	fbGetInputNotification(	bEnable := TRUE,
							eEventScheme := eEventScheme,
							nAddressInfo1 := nAddressInfo01,
							nAddressInfo2 := nAddressInfo02,
							nEventInfo => nInputValue);
	CASE fbGetInputNotification.nEventInfo OF
		0: sInputValue := 'Push button released';
		1: sInputValue := 'Push button pressed';
		2: sInputValue := 'Short press';
		5: sInputValue := 'Double press';
		9: sInputValue := 'Long press start';
		11: sInputValue := 'Long press repeat';
		12: sInputValue := 'Long press stop';
		14: sInputValue := 'Button free';
		15: sInputValue := 'Button stuck';
	END_CASE
{endregion}
{region "Read"}
5:
{region "Start Qiescent Mode"}
	fb103StartQuiescentMode(bStart := TRUE,
							eAddressType := Tc3_DALI.E_DALIAddressType.Broadcast,
							eCommandPriority := Tc3_DALI.E_DALICommandPriority.Middle);
	IF (NOT fb103StartQuiescentMode.bBusy) THEN
		fb103StartQuiescentMode(bStart := FALSE);
		nStep := 10;
	END_IF
{endregion}
10:
{region "Query Instance Error"}
	fb103QueryInstanceError(bStart := TRUE,
							nAddress := nAddress,
							eAddressType := Tc3_DALI.E_DALIAddressType.Short,
							nInstanceAddress := nInstanceAddress,
							eInstanceAddressType := Tc3_DALI.E_DALIInstanceAddressType.InstanceNumber,
							eCommandPriority := Tc3_DALI.E_DALICommandPriority.Middle,
							nInstanceError => nInstanceError);
	IF (NOT fb103QueryInstanceError.bBusy) THEN
		fb103QueryInstanceError(bStart := FALSE);
		nStep := 20;
	END_IF
{endregion}
20:
{region "Query Instance Status"}
	fb103QueryInstanceStatus(	bStart := TRUE,
								nAddress := nAddress,
								eAddressType := Tc3_DALI.E_DALIAddressType.Short,
								nInstanceAddress := nInstanceAddress,
								eInstanceAddressType := Tc3_DALI.E_DALIInstanceAddressType.InstanceNumber,
								eCommandPriority := Tc3_DALI.E_DALICommandPriority.Middle);
	IF (NOT fb103QueryInstanceStatus.bBusy) THEN
		fb103QueryInstanceStatus(bStart := FALSE);
		IF (fb103QueryInstanceStatus.nInstanceStatus.1) THEN
			bEnable := TRUE;
		END_IF
		nStep := 30;
	END_IF
30:
{region "Query Resolution"}
	fb103QueryResolution(	bStart := TRUE,
							nAddress := nAddress,
							eAddressType := Tc3_DALI.E_DALIAddressType.Short,
							nInstanceAddress := nInstanceAddress,
							eInstanceAddressType := Tc3_DALI.E_DALIInstanceAddressType.InstanceNumber,
							eCommandPriority := Tc3_DALI.E_DALICommandPriority.Middle,
							nResolution => nResolution);
	IF (NOT fb103QueryResolution.bBusy) THEN
		fb103QueryResolution(bStart := FALSE);
		nStep := 40;
	END_IF
{endregion}
40:
{region "Query Input Value"}
	fb103QueryInputValue(	bStart := TRUE,
							nAddress := nAddress,
							eAddressType := Tc3_DALI.E_DALIAddressType.Short,
							nInstanceAddress := nInstanceAddress,
							eInstanceAddressType := Tc3_DALI.E_DALIInstanceAddressType.InstanceNumber,
							eCommandPriority := Tc3_DALI.E_DALICommandPriority.Middle,
							nResolution := nResolution);
	IF (NOT fb103QueryInputValue.bBusy) THEN
		fb103QueryInputValue(bStart := FALSE);
		CASE fb103QueryInputValue.nInputValue OF
			0: sInputValue := 'Push button released';
			1: sInputValue := 'Push button pressed';
			2: sInputValue := 'Short press';
			5: sInputValue := 'Double press';
			9: sInputValue := 'Long press start';
			11: sInputValue := 'Long press repeat';
			12: sInputValue := 'Long press stop';
			14: sInputValue := 'Button free';
			15: sInputValue := 'Button stuck';
		END_CASE
		nStep := 50;
	END_IF
{endregion}
50:
{region "Query Event Scheme"}
	fb103QueryEventScheme(	bStart := TRUE,
							nAddress := nAddress,
							eAddressType := Tc3_DALI.E_DALIAddressType.Short,
							nInstanceAddress := nInstanceAddress,
							eInstanceAddressType := Tc3_DALI.E_DALIInstanceAddressType.InstanceNumber,
							eCommandPriority := Tc3_DALI.E_DALICommandPriority.Middle,
							eEventScheme => eEventScheme);
	IF (NOT fb103QueryEventScheme.bBusy) THEN
		fb103QueryEventScheme(bStart := FALSE);
		nStep := 60;
	END_IF
{endregion}
60:
{region "Query Event Filter"}
	fb103QueryEventFilter(	bStart := TRUE,
							nAddress := nAddress,
							eAddressType := Tc3_DALI.E_DALIAddressType.Short,
							nInstanceAddress := nInstanceAddress,
							eInstanceAddressType := Tc3_DALI.E_DALIInstanceAddressType.InstanceNumber,
							eCommandPriority := Tc3_DALI.E_DALICommandPriority.Middle,
							nEventFilter => nEventFilter);
	IF (NOT fb103QueryEventFilter.bBusy) THEN
		fb103QueryEventFilter(bStart := FALSE);
		bButtonReleased := nEventFilter.0;
		bButtonPressed := nEventFilter.1;
		bShortPress := nEventFilter.2;
		bDoublePress := nEventFilter.3;
		bLongPressStart := nEventFilter.4;
		bLongPressRepeat := nEventFilter.5;
		bLongPressStop := nEventFilter.6;
		bButtonStuck := nEventFilter.7;
		nStep := 70;
	END_IF
{endregion}
70:
{region "Query Repeat Timer"}
	fb301QueryRepeatTimer(	bStart := TRUE,
							nAddress := nAddress,
							eAddressType := Tc3_DALI.E_DALIAddressType.Short,
							nInstanceAddress := nInstanceAddress,
							eInstanceAddressType := Tc3_DALI.E_DALIInstanceAddressType.InstanceNumber,
							eCommandPriority := Tc3_DALI.E_DALICommandPriority.Middle);
	nRepeat := (fb301QueryRepeatTimer.nRepeat * 20);
	IF (NOT fb301QueryRepeatTimer.bBusy) THEN
		fb301QueryRepeatTimer(bStart := FALSE);
		nStep := 80;
	END_IF
{endregion}
80:
{region "Query Stuck Timer"}
	fb301QueryStuckTimer(	bStart := TRUE,
							nAddress := nAddress,
							eAddressType := Tc3_DALI.E_DALIAddressType.Short,
							nInstanceAddress := nInstanceAddress,
							eInstanceAddressType := Tc3_DALI.E_DALIInstanceAddressType.InstanceNumber,
							eCommandPriority := Tc3_DALI.E_DALICommandPriority.Middle,
							nStuck => nStuck);
	IF (NOT fb301QueryStuckTimer.bBusy) THEN
		fb301QueryStuckTimer(bStart := FALSE);
		nStep := 90;
	END_IF
{endregion}
90:
{region "Query Short Timer"}
	fb301QueryShortTimer(	bStart := TRUE,
							nAddress := nAddress,
							eAddressType := Tc3_DALI.E_DALIAddressType.Short,
							nInstanceAddress := nInstanceAddress,
							eInstanceAddressType := Tc3_DALI.E_DALIInstanceAddressType.InstanceNumber,
							eCommandPriority := Tc3_DALI.E_DALICommandPriority.Middle);
	nShort := (fb301QueryShortTimer.nShort * 20);
	IF (NOT fb301QueryShortTimer.bBusy) THEN
		fb301QueryShortTimer(bStart := FALSE);
		nStep := 95;
	END_IF
{endregion}
95:
{region "Query Short Timer Min"}
	fb301QueryShortTimerMin(bStart := TRUE,
							nAddress := nAddress,
							eAddressType := Tc3_DALI.E_DALIAddressType.Short,
							nInstanceAddress := nInstanceAddress,
							eInstanceAddressType := Tc3_DALI.E_DALIInstanceAddressType.InstanceNumber,
							eCommandPriority := Tc3_DALI.E_DALICommandPriority.Middle);
	nShortMin := (fb301QueryShortTimerMin.nShortMin * 20);
	IF (NOT fb301QueryShortTimerMin.bBusy) THEN
		fb301QueryShortTimerMin(bStart := FALSE);
		nStep := 100;
	END_IF
{endregion}
100:
{region "Query Double Timer"}
	fb301QueryDoubleTimer(	bStart := TRUE,
							nAddress := nAddress,
							eAddressType := Tc3_DALI.E_DALIAddressType.Short,
							nInstanceAddress := nInstanceAddress,
							eInstanceAddressType := Tc3_DALI.E_DALIInstanceAddressType.InstanceNumber,
							eCommandPriority := Tc3_DALI.E_DALICommandPriority.Middle);
	nDouble := (fb301QueryDoubleTimer.nDouble * 20);
	IF (NOT fb301QueryDoubleTimer.bBusy) THEN
		fb301QueryDoubleTimer(bStart := FALSE);
		nStep := 105;
	END_IF
{endregion}
105:
{region "Query Double Timer"}
	fb301QueryDoubleTimerMin(	bStart := TRUE,
								nAddress := nAddress,
								eAddressType := Tc3_DALI.E_DALIAddressType.Short,
								nInstanceAddress := nInstanceAddress,
								eInstanceAddressType := Tc3_DALI.E_DALIInstanceAddressType.InstanceNumber,
								eCommandPriority := Tc3_DALI.E_DALICommandPriority.Middle);
	nDoubleMin := (fb301QueryDoubleTimerMin.nDoubleMin * 20);
	IF (NOT fb301QueryDoubleTimerMin.bBusy) THEN
		fb301QueryDoubleTimerMin(bStart := FALSE);
		nStep := 110;
	END_IF
{endregion}
110:
{region "Query Event Priority"}
	fb103QueryEventPriority(bStart := TRUE,
							nAddress := nAddress,
							eAddressType := Tc3_DALI.E_DALIAddressType.Short,
							nInstanceAddress := nInstanceAddress,
							eInstanceAddressType := Tc3_DALI.E_DALIInstanceAddressType.InstanceNumber,
							eCommandPriority := Tc3_DALI.E_DALICommandPriority.Middle,
							eEventPriority => eEventPriority);
	IF (NOT fb103QueryEventPriority.bBusy) THEN
		fb103QueryEventPriority(bStart := FALSE);
		nStep := 120;
	END_IF 
{endregion}
120:
{region "Stop Qiescent Mode"}
	fb103StopQuiescentMode(	bStart := TRUE,
							eAddressType := Tc3_DALI.E_DALIAddressType.Broadcast,
							eCommandPriority := Tc3_DALI.E_DALICommandPriority.Middle);
	IF (NOT fb103StopQuiescentMode.bBusy) THEN
		fb103StopQuiescentMode(	bStart := FALSE);
		nStep := 0;
	END_IF
{endregion}
{endregion}
{region "Write"}
1000:
{region "Enable or Disable Instance"}
	IF (bEnable) THEN
		fb103EnableInstance(bStart := TRUE,
							nAddress := nAddress,
							eAddressType := Tc3_DALI.E_DALIAddressType.Short,
							nInstanceAddress := nInstanceAddress,
							eInstanceAddressType := Tc3_DALI.E_DALIInstanceAddressType.InstanceNumber,
							eCommandPriority := Tc3_DALI.E_DALICommandPriority.Middle);
		IF (NOT fb103EnableInstance.bBusy) THEN
			fb103EnableInstance(bStart := FALSE);
			nStep := 1010;
		END_IF
	ELSE
		fb103DisableInstance(	bStart := TRUE,
								nAddress := nAddress,
								eAddressType := Tc3_DALI.E_DALIAddressType.Short,
								nInstanceAddress := nInstanceAddress,
								eInstanceAddressType := Tc3_DALI.E_DALIInstanceAddressType.InstanceNumber,
								eCommandPriority := Tc3_DALI.E_DALICommandPriority.Middle);
		IF (NOT fb103DisableInstance.bBusy) THEN
			fb103DisableInstance(bStart := FALSE);
			nStep := 0;
		END_IF
	END_IF
{endregion}
1010:
{region "Set Event Scheme"}
	fb103SetEventScheme(bStart := TRUE,
						nAddress := nAddress,
						eAddressType := Tc3_DALI.E_DALIAddressType.Short,
						nInstanceAddress := nInstanceAddress,
						eInstanceAddressType := Tc3_DALI.E_DALIInstanceAddressType.InstanceNumber,
						eCommandPriority := Tc3_DALI.E_DALICommandPriority.Middle,
						eEventScheme := eEventScheme);
	IF (NOT fb103SetEventScheme.bBusy) THEN
		fb103SetEventScheme(bStart := FALSE);
		nStep := 1020;
	END_IF
{endregion}
1020:
{region "Set Event Filter"}
	nEventFilter.0 := bButtonReleased;
	nEventFilter.1 := bButtonPressed;
	nEventFilter.2 := bShortPress;
	nEventFilter.3 := bDoublePress;
	nEventFilter.4 := bLongPressStart;
	nEventFilter.5 := bLongPressRepeat;
	nEventFilter.6 := bLongPressStop;
	nEventFilter.7 := bButtonStuck;
	fb103SetEventFilter(bStart := TRUE,
						nAddress := nAddress,
						eAddressType := Tc3_DALI.E_DALIAddressType.Short,
						nInstanceAddress := nInstanceAddress,
						eInstanceAddressType := Tc3_DALI.E_DALIInstanceAddressType.InstanceNumber,
						eCommandPriority := Tc3_DALI.E_DALICommandPriority.Middle,
						nEventFilter := nEventFilter);
	IF (NOT fb103SetEventFilter.bBusy) THEN
		fb103SetEventFilter(bStart := FALSE);
		nStep := 1030;
	END_IF
{endregion}
1030:
{region "Set Repeat Timer"}
	IF (bNoRepeatTimer) THEN
		nStep := 1040;
	ELSE
		fb301SetRepeatTimer(bStart := TRUE,
							nAddress := nAddress,
							eAddressType := Tc3_DALI.E_DALIAddressType.Short,
							nInstanceAddress := nInstanceAddress,
							eInstanceAddressType := Tc3_DALI.E_DALIInstanceAddressType.InstanceNumber,
							eCommandPriority := Tc3_DALI.E_DALICommandPriority.Middle,
							nRepeat := TO_BYTE (nRepeat / 20));
		IF (NOT fb301SetRepeatTimer.bBusy) THEN
			fb301SetRepeatTimer(bStart := FALSE);
			nStep := 1040;
		END_IF
	END_IF
{endregion}
1040:
{region "Set Stuck Timer"}
	IF (bNoStuckTimer) THEN
		nStep := 1050;
	ELSE
		fb301SetStuckTimer(	bStart := TRUE,
							nAddress := nAddress,
							eAddressType := Tc3_DALI.E_DALIAddressType.Short,
							nInstanceAddress := nInstanceAddress,
							eInstanceAddressType := Tc3_DALI.E_DALIInstanceAddressType.InstanceNumber,
							eCommandPriority := Tc3_DALI.E_DALICommandPriority.Middle,
							nStuck := nStuck);
		IF (NOT fb301SetStuckTimer.bBusy) THEN
			fb301SetStuckTimer(bStart := FALSE);
			nStep := 1050;
		END_IF
	END_IF
{endregion}
1050:
{region "Set Short Timer"}
	IF (bNoShortTimer) THEN
		nStep := 1060;
	ELSE
		fb301SetShortTimer(	bStart := TRUE,
							nAddress := nAddress,
							eAddressType := Tc3_DALI.E_DALIAddressType.Short,
							nInstanceAddress := nInstanceAddress,
							eInstanceAddressType := Tc3_DALI.E_DALIInstanceAddressType.InstanceNumber,
							eCommandPriority := Tc3_DALI.E_DALICommandPriority.Middle,
							nShort := TO_BYTE(nShort / 20));
		IF (NOT fb301SetShortTimer.bBusy) THEN
			fb301SetShortTimer(bStart := FALSE);
			nStep := 1060;
		END_IF
	END_IF
{endregion}
1060:
{region "Set Double Timer"}
	IF (bNoDoubleTimer) THEN
		nStep := 1070;
	ELSE
		fb301SetDoubleTimer(bStart := TRUE,
							nAddress := nAddress,
							eAddressType := Tc3_DALI.E_DALIAddressType.Short,
							nInstanceAddress := nInstanceAddress,
							eInstanceAddressType := Tc3_DALI.E_DALIInstanceAddressType.InstanceNumber,
							eCommandPriority := Tc3_DALI.E_DALICommandPriority.Middle,
							nDouble := TO_BYTE(nDouble / 20));
		IF (NOT fb301SetDoubleTimer.bBusy) THEN
			fb301SetDoubleTimer(bStart := FALSE);
			nStep := 1070;
		END_IF
	END_IF
1070:
{region "Set Event Priority"}
	fb103SetEventPriority(	bStart := TRUE,
							nAddress := nAddress,
							eAddressType := Tc3_DALI.E_DALIAddressType.Short,
							nInstanceAddress := nInstanceAddress,
							eInstanceAddressType := Tc3_DALI.E_DALIInstanceAddressType.InstanceNumber,
							eCommandPriority := Tc3_DALI.E_DALICommandPriority.Middle,
							eEventPriority := eEventPriority);
	IF (NOT fb103SetEventPriority.bBusy) THEN
		fb103SetEventPriority(bStart := FALSE);
		nStep := 0;
	END_IF
{endregion}
END_CASE
{endregion}
{endregion}

END_FUNCTION_BLOCK

// ---- POUs/DALI/DALI_Setup/FBs/GearType.TcPOU
FUNCTION GearType : STRING[80]
VAR_INPUT
	nGearType	:	BYTE;
END_VAR
VAR
	i: INT;
	aText	:	ARRAY [0..7] OF STRING[80];
END_VAR

GearType := '';
	aText[0] := 'Output is an electronic switch';
	aText[1] := 'Output is a relay with default open contacts';
	aText[2] := 'Output is a relay with default closed contacts';
	aText[3] := 'Output has a transient suppressor';
	aText[4] := 'Load inrush current limitation is integrated';
	aText[5] := '';
	aText[6] := '';
	aText[7] := '';
FOR i := 0 TO 7 DO
	IF nGearType.0 THEN
		GearType := aText[i];
	ELSE
		GearType := '';
	END_IF
	nGearType := ROR (nGearType,1);
END_FOR

IF (nGearType.1 AND nGearType.2)	THEN 
	GearType := 'Latched Output, the latched state does not change when power is removed';
END_IF

END_FUNCTION

// ---- POUs/DALI/PRGs/EnergyData/P_DALI_Energy_Line.TcPOU
(*
EnergyReporting reads ActiveEnergy (part 252) for all present ballasts on all (configured) DALI-lines where GVL_DALI.g_arrEnergyData[*DALI-line*,*ballast*].bHasEnergyData is TRUE.
Results are stored in GVL_DALI.g_arrEnergyData[*DALI-line*,*ballast*].fActiveEnergy. Energy Data for individual ballasts is NOT persistent.
The engergy sum per DALI-Line (Wh) and Total Energy (kWh) are persistent.

If bCheckActiveEnergy is TRUE, all present ballasts are queried for ActiveEnergy and bHasEnergyData is updated accordingly.
This will result in errors for any ballast that does not comply with part 252.
Errors will not be triggered for activations where bCheckActiveEnergy is FALSE.

After shutdown or download to PLC EnergyReporting is activated automatically internally with bCheckActiveEnergy set to TRUE

EnergyReporting is activated automatically at TOD 0:00, 6:00, 12:00, 18:00 (configurable)

NB:	The priority of commands are set to "middle" internally. Updating all lines will take a couple of minutes to finish, so be patient.
	Other critical commands on the DALI-lines take priotity.
	Add appropriate communication immediately after configuration of a new KL6821 terminal.
	That is, arrfbDALI_EnergyReporting[*DALI-Line*].ipDALICommunication := P_DALI_Background.arrfbKL6821Communication[*DALI-Line*];
*)


PROGRAM P_DALI_Energy_Line
VAR
	arrfbDALI_EnergyReporting	: ARRAY[1..SH_Light.DALI_Param.MAX_DALIV2_LINES] OF FB_DALI_EnergyReporting;
	fbDALI_EnergyDataManagement	: SH_Light.FB_DALI_EnergyDataManagement;
	nNumOfEnergyLines			: BYTE;
	bReadEnergyDataAllLines		: BOOL;
	bReportingDone				: BOOL;
	fbRTrig_ReportingDone		: R_TRIG;
	bRTrigReportingDone			: BOOL;
	
	//Task scheduling
	stLocalSystemTime 		: TIMESTRUCT;
	fbLocalSystemTime 		: FB_LocalSystemTime;
	bGetTime 				: BOOL := TRUE;
	tTimeOut 				: TIME := DEFAULT_ADS_TIMEOUT;
	bLocalSystemTimeValid	: BOOL;
	tzID       				: E_TimeZoneID := eTimeZoneID_Invalid;
	
	tdSystemTime			: TOD;
	btestTodCompare			: BOOL;
	
	
END_VAR
VAR CONSTANT
	tdMidnight						: TOD := TOD#0:0:0;
	tdMorning						: TOD := TOD#6:0:0;
	tdMidDay						: TOD := TOD#12:0:0;
	tdEvening						: TOD := TOD#18:0:0;
	tCheckDuration					: TIME:= T#5S;
	tdTestsum						: TOD := (tdMidnight + tCheckDuration);
END_VAR

VAR PERSISTENT
	arrDaliLineEnergySumWh				: ARRAY[1..SH_Light.DALI_Param.MAX_DALIV2_LINES] OF LREAL;
	fTotalEnergyWh						: LREAL;
	nMaxControlGearOperatingHours		: UINT;
END_VAR


arrfbDALI_EnergyReporting[1].ipDALICommunication := P_DALI_Background.arrfbKL6821Communication[1];
arrfbDALI_EnergyReporting[2].ipDALICommunication := P_DALI_Background.arrfbKL6821Communication[2];
arrfbDALI_EnergyReporting[3].ipDALICommunication := P_DALI_Background.arrfbKL6821Communication[3];
arrfbDALI_EnergyReporting[4].ipDALICommunication := P_DALI_Background.arrfbKL6821Communication[4];
//arrfbDALI_EnergyReporting[5].ipDALICommunication := P_DALI_Background.arrfbKL6821Communication[5];
//arrfbDALI_EnergyReporting[6].ipDALICommunication := P_DALI_Background.arrfbKL6821Communication[6]; // for more update SH_Light.DALI_Param.MAX_DALIV2_LINES

nNumOfEnergyLines := 4;

fbLocalSystemTime(
	sNetID:= '', 
	bEnable:= bGetTime, 
	dwCycle:= 2, // cycle time (in seconds) , Synchronization  every 2 seconds.
	dwOpt:= 1, //Bit 0: If this is set, the Windows system time is additionally synchronized cyclically with the hardware clock (RTC) (corresponds to the function NT_SetTimeToRTCTime).
	tTimeout:= tTimeOut, 
	bValid=> bLocalSystemTimeValid, 
	systemTime=> stLocalSystemTime, 
	tzID=> tzID);
	
tdSystemTime := SYSTEMTIME_TO_TOD(systemTime := stLocalSystemTime);
IF	((tdSystemTime > tdMidnight AND tdSystemTime < (tdMidnight + tCheckDuration)) OR (tdSystemTime > tdMorning AND tdSystemTime < (tdMorning + tCheckDuration)) OR
	(tdSystemTime > tdMidDay AND tdSystemTime < (tdMidDay + tCheckDuration)) OR (tdSystemTime > tdEvening AND tdSystemTime < (tdEvening + tCheckDuration))) THEN
	bReadEnergyDataAllLines := TRUE;
END_IF

fbDALI_EnergyDataManagement(
	NumOfEnergyLines				:= nNumOfEnergyLines,
	bReadEnergyDataAllLines 		:= bReadEnergyDataAllLines,
	arrfbDALI_EnergyReporting		:= arrfbDALI_EnergyReporting,
	arrDaliLineEnergySum			:= arrDaliLineEnergySumWH,
	fTotalEnergyWh					:= fTotalEnergyWh,
	nMaxControlGearOperatingHours	:= nMaxControlGearOperatingHours,
	bReportingDone					=> bReportingDone
);
GVL_AHDataModbus.nTotalEnergy10kWh := TO_UINT(TRUNC(fTotalEnergyWh*EXPT(10,-4)));  //FB_DALI_EnergyDataManagement makes sure only positive values are returned. As so, conversion from REAL to UINT is appropriate
GVL_AHDataModbus.nMaxControlGearOperatingHours := nMaxControlGearOperatingHours;

END_PROGRAM

// ---- POUs/EnOcean/P_EnOcean.TcPOU
PROGRAM P_EnOcean
VAR
	fbKL6581			: FB_KL6581;
	stKL6581_in  AT %I* : KL6581_INPUT;
	stKL6581_out AT %Q*	: KL6581_OUTPUT;
	stKL6581			: STR_KL6581;
	bInitCom			: BOOL := TRUE;
	
	arrEnOcean_Search	: ARRAY [1..8] OF FB_EnOcean_Search;
	nSearchIdx			: BYTE;
	bSerach				: BOOL;
	arrDevices			: ARRAY [1..8] OF INT;
	arrID				: ARRAY [1..8, 0..255] OF DWORD;
	
		//Trykknapper Atrium
	fbAtriumNiveau_Tryk_PladeB				: FB_Rec_RPS_Switch;
	fbAtriumNiveau_Tryk_Sevice				: FB_Rec_RPS_Switch;			

	//Trykknapper på gange

	
	//Trykknapper i rum
	fbRum_4_424_Tryk						: FB_Rec_RPS_Switch;
	fbRum_4_426_Tryk						: FB_Rec_RPS_Switch;
	fbRum_5_441A_Tryk						: FB_Rec_RPS_Switch;
	fbGang_5_441B_Tryk						: FB_Rec_RPS_Switch;
	fbRum_5_444_Tryk						: FB_Rec_RPS_Switch;
	fbRum_5_448A_Tryk						: FB_Rec_RPS_Switch;
	fbRum_5_450_Tryk						: FB_Rec_RPS_Switch;	
	fbRum_5_452_Tryk						: FB_Rec_RPS_Switch;
	fbRum_5_454_Tryk						: FB_Rec_RPS_Switch;
	fbRum_5_411C_Tryk						: FB_Rec_RPS_Switch;
END_VAR

VAR CONSTANT
	byNode_1: BYTE := 1;
	byNode_2: BYTE := 2;
	byNode_3: BYTE := 3;
	byNode_4: BYTE := 4;
	byNode_5: BYTE := 5;
	byNode_6: BYTE := 6;
	byNode_7: BYTE := 7;
	byNode_8: BYTE := 8;
END_VAR


(* Kommunikation mit der KL6581. *)
(* Communication with the KL6581. *)
fbKL6581(
	bInit			:= bInitCom,
	nIdx			:= 2,
	stKL6581_in		:= stKL6581_In,
	stKL6581_out	:= stKL6581_Out,
	bReady			=> ,
	bBusy			=> ,
	bError			=> ,
	iErrorID		=> ,
	str_KL6581		=> stKL6581);

GVL_AHDataModbus.EnOceanError	:= TO_UINT(fbKL6581.iErrorID);
(* Warten bis der Kommunikationsbaustein initialisiert wurde.*)
(* Wait until the communication function block has been initialized. *)
IF (NOT fbKL6581.bReady) THEN
	RETURN;
END_IF

FOR nSearchIdx:= 1 TO 8 DO
	arrEnOcean_Search[nSearchIdx](
		bStart:= TRUE, 
		str_KL6581:= stKL6581 , 
		byNode:= nSearchIdx, 
		bReceive=> , 
		iDevices=>arrDevices[nSearchIdx] , 
		ar_ID=> );
		
		MEMCPY(ADR(arrID[nSearchIdx,0]), ADR(arrEnOcean_Search[nSearchIdx].ar_ID), SIZEOF(arrEnOcean_Search[nSearchIdx].ar_ID)); 
END_FOR

//Gange



//RUM
 //
P_Rum_4_424();
P_Rum_4_426();
P_Rum_5_441A();
P_Gang_5_441B();
P_Rum_5_444();
P_Rum_5_448A();
P_Rum_5_450();
P_Rum_5_452();
P_Rum_5_454();
P_Rum_5_411C();
//AtriumNiveau
A_AtriumNiveau();

ACTION A_AtriumNiveau:
fbAtriumNiveau_Tryk_PladeB(
	str_KL6581:=stKL6581 , 
	byNode:=0, 
	dw_ID:= 16#0029B92D, 
	str_EnOceanSwitch=> GVL_EnOcean.strEnOceanSwitch_AtriumNiveau_PladeB,
	by_Node=> , 
	bReceive=> );

//knap 2 
(*
fbAtriumNiveau_Tryk_Sevice(
	str_KL6581:=stKL6581 , 
	byNode:=0, 
	dw_ID:= 16#00FEE4FE87, 
	str_EnOceanSwitch=> GVL_EnOcean.strEnOceanSwitch_AtriumNiveau_Service, 
	by_Node=> , 
	bReceive=> );
*)
END_ACTION

ACTION P_Gang_5_441B:
fbGang_5_441B_Tryk(
	str_KL6581:=stKL6581 , 
	byNode:=4 , 
	dw_ID:=  16#002A0890, 
	str_EnOceanSwitch=> GVL_EnOcean.strEnOceanSwitch_Gang_5_441B, 
	by_Node=> , 
	bReceive=> );
END_ACTION

ACTION P_Rum_4_424:
fbRum_4_424_Tryk(
	str_KL6581:=stKL6581 , 
	byNode:=2 , 
	dw_ID:= 16#0029AB88, 
	str_EnOceanSwitch=> GVL_EnOcean.strEnOceanSwitch_Rum_4_424, 
	by_Node=> , 
	bReceive=> );
END_ACTION

ACTION P_Rum_4_426:
fbRum_4_426_Tryk(
	str_KL6581:=stKL6581 , 
	byNode:=2 , 
	dw_ID:= 16#0029AAD6, 
	str_EnOceanSwitch=> GVL_EnOcean.strEnOceanSwitch_Rum_4_426, 
	by_Node=> , 
	bReceive=> );
END_ACTION

ACTION P_Rum_5_411C:
fbRum_5_411C_Tryk(
	str_KL6581:=stKL6581 , 
	byNode:=4 , 
	dw_ID:=  16#0029AD43, 
	str_EnOceanSwitch=> GVL_EnOcean.strEnOceanSwitch_Rum_5_411C, 
	by_Node=> , 
	bReceive=> );
END_ACTION

ACTION P_Rum_5_441A:
fbRum_5_441A_Tryk(
	str_KL6581:=stKL6581 , 
	byNode:=4 , 
	dw_ID:=  16#00290EC2, 
	str_EnOceanSwitch=> GVL_EnOcean.strEnOceanSwitch_Rum_5_441A, 
	by_Node=> , 
	bReceive=> );
END_ACTION

ACTION P_Rum_5_444:
fbRum_5_444_Tryk(
	str_KL6581:=stKL6581 , 
	byNode:=4 , 
	dw_ID:=  16#0029B74E, 
	str_EnOceanSwitch=> GVL_EnOcean.strEnOceanSwitch_Rum_5_444, 
	by_Node=> , 
	bReceive=> );
END_ACTION

ACTION P_Rum_5_448A:
fbRum_5_448A_Tryk(
	str_KL6581:=stKL6581 , 
	byNode:=4 , 
	dw_ID:=  16#0029AB8B, 
	str_EnOceanSwitch=> GVL_EnOcean.strEnOceanSwitch_Rum_5_448A, 
	by_Node=> , 
	bReceive=> );
END_ACTION

ACTION P_Rum_5_450:
fbRum_5_450_Tryk(
	str_KL6581:=stKL6581 , 
	byNode:=4 , 
	dw_ID:=  16#0029ABB9, 
	str_EnOceanSwitch=> GVL_EnOcean.strEnOceanSwitch_Rum_5_450, 
	by_Node=> , 
	bReceive=> );
END_ACTION

ACTION P_Rum_5_452:
fbRum_5_452_Tryk(
	str_KL6581:=stKL6581 , 
	byNode:=4 , 
	dw_ID:=  16#0029B8D2, 
	str_EnOceanSwitch=> GVL_EnOcean.strEnOceanSwitch_Rum_5_452, 
	by_Node=> , 
	bReceive=> );
END_ACTION

ACTION P_Rum_5_454:
fbRum_5_454_Tryk(
	str_KL6581:=stKL6581 , 
	byNode:=4 , 
	dw_ID:=  16#0029B75D, 
	str_EnOceanSwitch=> GVL_EnOcean.strEnOceanSwitch_Rum_5_454, 
	by_Node=> , 
	bReceive=> );
END_ACTION

END_PROGRAM

// ---- POUs/MAIN.TcPOU
PROGRAM MAIN
VAR
	nAlive: INT;
	breset: BOOL;
	nDemoVariable : INT;
	nCX8200_State	AT %I*	: UINT;
	P_Rum_6_217: INT;
END_VAR

VAR PERSISTENT
	nDemoVar_Persist: INT;
END_VAR

nAlive:= nAlive + 1;
GVL_AHDataModbus.nCX8200_State_MB := nCX8200_State;

P_SystemDK.M_nCyclic(bReset := breset );
P_DALI_DIAG();
DALI_Commissioning();
P_DALI_Energy_Line();
P_AHModbusComm();


//Gange
P_Gang_4_413();
P_Gang_5_441B();
P_gang_7_401();
P_Gang_4_434A();
P_gang_5_441();


//Rum
P_Rum_4_426();
P_Rum_4_424();

P_rum_5_441A();
P_Rum_5_411C();
P_Rum_5_444();
P_Rum_5_448A();
P_Rum_5_448B();
P_Rum_5_450B();
P_Rum_5_450();
P_Rum_5_452();
P_Rum_5_454();
P_Rum_5_456();


//Testprogrammer
//P_DALI_Energy_Firmware_Test();

END_PROGRAM

// ---- GlobalTextList.TcGTLO
TEXTLIST GlobalTextList
  3955 = ' %5.2f h'
  1376 = ' %d %%'
  307 = ' %d days'
  1111 = '%2.1f  mA'
  102 = '%5.1f W'
  269 = '%5.2f h'
  621 = '%d'
  1617 = '%d %%'
  2081 = '%d days'
  3200 = '%d h'
  1372 = '%d Hz'
  2105 = '%d min'
  2025 = '%d ms'
  1540 = '%d s'
  1613 = '%d V'
  2272 = '%d weeks'
  1359 = '%d °C'
  376 = '%s'
  640 = '0'
  641 = '1'
  661 = '10'
  662 = '11'
  663 = '12'
  999 = '13'
  1000 = '14'
  1001 = '15'
  1002 = '16'
  1003 = '17'
  1004 = '18'
  1005 = '19'
  195 = '2'
  1006 = '20'
  1007 = '21'
  1008 = '22'
  1009 = '23'
  1010 = '24'
  1011 = '25'
  1012 = '26'
  1013 = '27'
  1014 = '28'
  1015 = '29'
  654 = '3'
  1016 = '30'
  1017 = '31'
  1018 = '32'
  1019 = '33'
  1020 = '34'
  1021 = '35'
  1022 = '36'
  1023 = '37'
  1024 = '38'
  1025 = '39'
  655 = '4'
  1026 = '40'
  1027 = '41'
  1028 = '42'
  1029 = '43'
  1030 = '44'
  1031 = '45'
  1032 = '46'
  1033 = '47'
  1034 = '48'
  1035 = '49'
  656 = '5'
  358 = '50'
  359 = '51'
  360 = '52'
  361 = '53'
  362 = '54'
  363 = '55'
  364 = '56'
  365 = '57'
  366 = '58'
  367 = '59'
  657 = '6'
  368 = '60'
  369 = '61'
  370 = '62'
  371 = '63'
  658 = '7'
  659 = '8'
  660 = '9'
  1089 = 'AC-supply possible'
  644 = 'Actual Level:'
  650 = 'Address Type'
  236 = 'Addressing Per Physical Selection Supported'
  1533 = 'Adjustable Emergency Level'
  1175 = 'AM Operation active:'
  1044 = 'AM operation possible'
  1045 = 'Auto Test Capability'
  1799 = 'Battery Charge'
  710 = 'Battery Duration Failure'
  3347 = 'Battery Failure'
  3316 = 'Battery Fully Charged'
  2471 = 'Bit 0'
  379 = 'Bit 1'
  2734 = 'Bit 2'
  2320 = 'Bit 3'
  929 = 'Bit 4'
  2576 = 'Bit 5'
  2065 = 'Bit 6'
  1623 = 'Bit 7'
  6 = 'Bottom Button'
  471 = 'Broadcast'
  482 = 'Button 1'
  720 = 'Button 2'
  515 = 'Button pressed'
  498 = 'Button released'
  527 = 'Button stuck / free'
  3304 = 'Cancel Hold Timer'
  2101 = 'Catch Movement'
  2319 = 'Catching:'
  897 = 'Change Addresses'
  1971 = 'Checkbox'
  372 = 'Choose group:'
  98 = 'Choose scene:'
  1571 = 'Circuit Failure'
  1538 = 'Commands'
  618 = 'Complete new installation \n(all addresses will be removed)'
  807 = 'Control'
  645 = 'Control Gear Failure:'
  445 = 'Current protection active:'
  1716 = 'Current protection device'
  668 = 'Current protection enabled:'
  5 = 'Current Protector Enabled '
  1902 = 'DALI Line:'
  1135 = 'DC-supply possible'
  560 = 'Deadtime Timer:'
  1180 = 'DI1 falling edge'
  1218 = 'DI1 rising edge'
  1726 = 'DI2 falling edge'
  1876 = 'DI2 rising edge'
  519 = 'Dim Dwn'
  63 = 'Dim Up'
  2002 = 'Dimmer Temperature'
  936 = 'Dimming Curve:'
  1317 = 'Dimming method bit 0'
  776 = 'Dimming method bit 1'
  2135 = 'Do not lock process image in case of \nDALI commands from DI1 or DI2'
  4011 = 'Double press'
  1112 = 'Double Timer Min:'
  3936 = 'Double Timer:'
  811 = 'Down'
  594 = 'Down Switch-Off Threshold'
  2357 = 'Down Switch-On Threshold'
  1482 = 'Duration Test Delay Time'
  3527 = 'Duration Test Done And Result Valid'
  3086 = 'Duration Test Failed'
  3077 = 'Duration Test Interval'
  2631 = 'Duration Test Is In Progress'
  2791 = 'Duration Test Max. Delay Exceed'
  1708 = 'Duration Test Request Pending'
  2905 = 'Duration Test Result'
  1759 = 'Emergency Lamp Failure'
  779 = 'Emergency Level'
  3733 = 'Emergency MaxLevel'
  3168 = 'Emergency Min Level'
  1204 = 'Emergency Mode'
  971 = 'Emergency Mode Active'
  1901 = 'Emergency Status'
  486 = 'Enable'
  828 = 'Enable:'
  1982 = 'EventPriority'
  32 = 'EventPriority:'
  494 = 'EventScheme'
  1113 = 'EventScheme:'
  125 = 'Extended Emergency Mode Active'
  1841 = 'Extended Fade Time only valid if Fade Time equals 0!'
  3956 = 'Extended Version'
  649 = 'Fade Running:'
  1074 = 'FadeRate'
  1079 = 'FadeTime'
  1610 = 'Failure Status'
  319 = 'Fast Fade Time:'
  2099 = 'Features'
  672 = 'Features (Read only)'
  206 = 'Features Byte 1'
  377 = 'Features Byte 2'
  2876 = 'Features Byte 3'
  3334 = 'Function Test Delay Time'
  3242 = 'Function Test Done And Result Valid'
  2712 = 'Function Test Failed'
  1801 = 'Function Test Interval'
  1945 = 'Function Test Is In Progress'
  3448 = 'Function Test Max. Delay Exceed'
  165 = 'Function Test Request Pending'
  967 = 'Gang 1.312A'
  256 = 'Gang 1.315'
  906 = 'Gang 1.316'
  207 = 'Gang 2.344'
  66 = 'Gang 2.344A'
  583 = 'Gang 2.350'
  985 = 'Gang 3.362A'
  67 = 'Gang 3.363A'
  173 = 'Gang 3.363B'
  406 = 'Gang 4.308'
  459 = 'Gang 4.330'
  327 = 'Gang 5.338'
  524 = 'Gang 6.310'
  316 = 'Gang 7.301'
  3204 = 'Gear Type'
  1409 = 'GearType'
  815 = 'Go to Scene'
  99 = 'Go to scene'
  468 = 'Group Address'
  2361 = 'Hardwired Inhibit Is Active'
  3553 = 'Hardwired Inhibit Supported'
  2225 = 'Hardwired Switch Is On'
  568 = 'Hold Timer:'
  199 = 'Hysteresis Min:'
  200 = 'Hysteresis:'
  790 = 'Identification Active'
  315 = 'Illuminance Level'
  37 = 'Inhibit'
  3340 = 'Inhibit Mode'
  540 = 'Input Value:'
  544 = 'Instance Error:'
  2895 = 'Instance Number:'
  3047 = 'Integral Control Gear'
  492 = 'Internal DALI power supply disabled'
  1771 = 'K-Bus Watchdog'
  3636 = 'Lamp Emergency Time'
  647 = 'Lamp Failure:'
  2812 = 'Lamp Total Operation Time'
  1521 = 'Leading Edge Mode Running'
  506 = 'LED module integrated'
  2077 = 'Linear Dimming Curve Active'
  2179 = 'Load current can be queried '
  1266 = 'Load Current Overload'
  1355 = 'Load current overload with output \nlevel reduction can be queried'
  306 = 'Load Decrease:'
  1137 = 'Load Increase:'
  2313 = 'Load over-current can be queried'
  2518 = 'Load Over-Current Shutdown'
  1226 = 'Load Rating'
  2963 = 'Load rating can be queried'
  2785 = 'Load unsuitable can be queried'
  1454 = 'Load voltage can be queried'
  516 = 'Load Voltage Out Of Limits'
  1811 = 'Lockable bytes: changeable if "Offset 2" has the Value 85 (0x55).\nFor changing use decimal value.'
  523 = 'Long press repeat'
  507 = 'Long press start'
  511 = 'Long press stop'
  43 = 'Lys Auto'
  444 = 'Lys Rum'
  489 = 'Lys Zone 1'
  2032 = 'Maintained Control Gear'
  2046 = 'Memory Bank:'
  3290 = 'Movement'
  531 = 'na'
  23 = 'Name'
  926 = 'Name of byte in memory bank'
  729 = 'NewAddress'
  588 = 'No Movement'
  1061 = 'Non-logarithmic dimming curve can \nbe selected'
  1795 = 'Normal Mode Active'
  572 = 'Occupied'
  808 = 'Off'
  22 = 'Offset'
  1329 = 'Offset in memory bank'
  726 = 'OldAddress'
  816 = 'On and Step Up'
  1207 = 'Open circuit detection can be queried'
  277 = 'Open Circuit:'
  1375 = 'Open Ciruit (No Load) Detect'
  619 = 'Optical feedback'
  963 = 'Output is current controlled'
  844 = 'Output regulated by current:'
  1545 = 'Parameters'
  2547 = 'Parameters Absolute Input Device'
  1580 = 'Parameters Generic Instance'
  78 = 'Parameters LED'
  309 = 'Parameters Light Sensor'
  556 = 'Parameters Occupancy Sensor'
  465 = 'Parameters Pushbutton Sensor'
  3234 = 'Physical Selection Supported'
  1847 = 'Physical selection supported'
  708 = 'PIR'
  457 = 'PIR status'
  1071 = 'Please check if Current Protector is present \nby reading parameters first.'
  308 = 'Please select the desired Short Address in the table above.'
  1458 = 'Please select the function you need from dropdown above'
  751 = 'Position Event'
  245 = 'Possible Operating Modes'
  719 = 'Power pulse operation'
  1744 = 'Power supply integrated'
  1561 = 'PP Operation active:'
  2321 = 'Prolong Time (30sec / Step)'
  970 = 'PWM Operation active:'
  1882 = 'PWM operation possible'
  1487 = 'Query idle time detection \nenabled'
  701 = 'Query load decrease enabled'
  1351 = 'Query load increase enabled'
  837 = 'Query reduction luminous flux \nregarding thermal overload'
  463 = 'Query short circuit enabled'
  1293 = 'Query thermal switch enabled'
  617 = 'Random Addressing'
  2174 = 'Rated Duration'
  881 = 'Re-Light / Reset Inhibit'
  373 = 'Read'
  1611 = 'Read Only'
  1531 = 'Reads all Fading Parameters'
  768 = 'Real Load Power'
  854 = 'Real load power can be queried'
  810 = 'Recall Max Level'
  809 = 'Recall Min Level'
  186 = 'Ref. Measurement failed:'
  439 = 'Reference System Power'
  2713 = 'Relight Rest Mode Supported'
  580 = 'Repeat'
  470 = 'Repeat Timer:'
  1913 = 'Report Timer:'
  716 = 'Reset Duration Test Done Flag'
  592 = 'Reset Function Test Done Flag'
  2418 = 'Reset inactive process image'
  3150 = 'Reset Lamp Time'
  648 = 'Reset State:'
  2888 = 'Resolution:'
  299 = 'Rest'
  591 = 'Rest Mode Active'
  2001 = 'RMS Load Current'
  784 = 'RMS Load Voltage'
  586 = 'RMS Supply Voltage'
  874 = 'Rum 1.106'
  65 = 'Rum 1.108'
  175 = 'Rum 1.111A'
  924 = 'Rum 1.111C'
  219 = 'Rum 1.111D'
  690 = 'Rum 1.111E'
  912 = 'Rum 1.115'
  126 = 'Rum 1.118'
  215 = 'Rum 1.312A'
  725 = 'Rum 1.318'
  839 = 'Rum 1.319'
  456 = 'Rum 1.320'
  800 = 'Rum 1.321'
  622 = 'Rum 1.322'
  646 = 'Rum 1.323'
  966 = 'Rum 1.324'
  95 = 'Rum 1.325'
  335 = 'Rum 1.326'
  150 = 'Rum 1.327'
  651 = 'Rum 1.328'
  980 = 'Rum 1.330'
  262 = 'Rum 1115'
  642 = 'Rum 2.341'
  978 = 'Rum 2.345'
  736 = 'Rum 2.349'
  593 = 'Rum 2.351'
  122 = 'Rum 2.352'
  27 = 'Rum 2.353'
  41 = 'Rum 2.354'
  697 = 'Rum 2.355'
  826 = 'Rum 2.356'
  561 = 'Rum 2.357'
  415 = 'Rum 3.365'
  981 = 'Rum 3.366'
  865 = 'Rum 3.367'
  212 = 'Rum 3.368'
  921 = 'Rum 3.369'
  329 = 'Rum 3.370'
  2134 = 'Rum 5.356'
  15 = 'Rum 5_352'
  430 = 'Rum 6.310 Sofagruppe'
  348 = 'Rum 6.327'
  891 = 'Rum 6.328'
  11 = 'Rum 6.329'
  72 = 'Rum 6.330B'
  197 = 'Rum 6.331'
  564 = 'Rum 6.333'
  997 = 'Rum 6.337'
  31 = 'Rum 6_330A'
  616 = 'Scan devices by address'
  1036 = 'Scene Level'
  814 = 'Scene:'
  1366 = 'Set Extended Fade Time'
  252 = 'Set Fade Rate'
  1875 = 'Set Fade Time'
  464 = 'Short Address'
  1090 = 'Short Address Range'
  1041 = 'Short Address:'
  34 = 'Short Circuit:'
  503 = 'Short press'
  1516 = 'Short Timer Min:'
  478 = 'Short Timer:'
  2548 = 'Shutdown Invalid Dimming Method'
  1085 = 'Single Short Address'
  395 = 'SP_Lux: %.0f'
  525 = 'SP_Lux: %f'
  615 = 'Start'
  582 = 'Start Duration Test'
  2374 = 'Start Function Test'
  155 = 'Start Identification'
  620 = 'Start with address:'
  2346 = 'State Incandescent Lamp'
  643 = 'Status'
  958 = 'Status Absolute Input Device'
  2506 = 'Status Generic Instance'
  77 = 'Status LED'
  317 = 'Status Light Sensor'
  597 = 'Status Occupancy Sensor'
  536 = 'Status Pushbutton Sensor'
  558 = 'Step Down'
  813 = 'Step Down and Off'
  818 = 'Step Up'
  1193 = 'Stop Test'
  164 = 'Stuck Timer:'
  1256 = 'Supply Frequency'
  2271 = 'Supply frequency can be queried'
  1975 = 'Supply Frequency Out of Limits'
  2505 = 'Supply voltage can be queried'
  2707 = 'Supply Voltage Out Of Limits'
  1042 = 'Switch Off'
  375 = 'Switch On'
  3781 = 'Switched Maintained Control Gear'
  2168 = 'Temperature can be queried'
  2458 = 'Terminal Event'
  1848 = 'Test Execution Timeout'
  849 = 'Test Type A'
  2013 = 'Thermal Overload'
  2042 = 'Thermal Overload with output\nlevel reduction can be queried'
  1108 = 'Thermal Overload:'
  355 = 'Thermal Shut Down:'
  2507 = 'Thermal Shutdown'
  2226 = 'Thermal Shutdown can be queried'
  2733 = 'Threshold Editable'
  305 = 'To'
  973 = 'Top Button'
  136 = 'Trailing Edge ModeRunning'
  475 = 'Unaddressed'
  817 = 'Up'
  3123 = 'Up Switch-Off Threshold'
  1449 = 'Up Switch-On Threshold'
  2521 = 'V%s'
  576 = 'Vacant'
  1205 = 'Value'
  24 = 'Value Dec'
  1435 = 'Value decimal'
  25 = 'Value Hex'
  2231 = 'Value hexadecimal,\nto change use\nvalue decimal'
  374 = 'Write'
  2104 = 'Write\nDimming Curve'
  1047 = 'Write default values'
  490 = 'Write parameters'
END_TEXTLIST

// ---- POUs/Alle_Rum/Gange/Gang_4_434A/Visualization_4_330_1_1_1_1_2.TcVIS
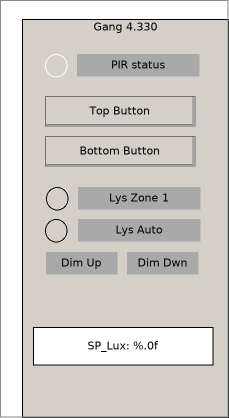
VISUALIZATION Visualization_4_330_1_1_1_1_2  // 229x418
    RoundedRectangle (22,19 207x399), "Gang 4.330"
    Rectangle (33,327 180x38), "SP_Lux: %.0f", text variable: P_Gang_5_135A.arrfbLysGruppe[1].fbLightCtrl.fLuxZone1
    Button (45,96 150x30), "Top Button"
        tap P_Gang_5_135A.bTopButtonZone1_Visu
    Button (45,136 150x30), "Bottom Button"
        tap P_Gang_5_135A.bBottomButtonZone1_Visu
    Ellipse (46,187 22x23), colour toggle: P_Gang_5_135A.fbLys.fbLightCtrl.bOnZone1
    Rectangle (78,187 122x22), "Lys Zone 1"
    Rectangle (46,252 71x22), "Dim Up", colour toggle: P_Gang_5_135A.arrfbLysGruppe[1].fbLightCtrl.bDimUp
    Rectangle (127,252 71x22), "Dim Dwn", colour toggle: P_Gang_5_135A.arrfbLysGruppe[1].fbLightCtrl.bDimDwn
    Ellipse (45,219 22x23), colour toggle: P_Gang_5_135A.arrfbLysGruppe[1].fbLightCtrl.bAutoZone1
    Rectangle (78,219 122x22), "Lys Auto"
    Ellipse (45,54 22x23), colour toggle: P_Gang_5_135A.arrfbLysGruppe[1].fbLightCtrl.bPIR
    Rectangle (77,54 122x22), "PIR status"
END_VISUALIZATION

// ---- POUs/Alle_Rum/Rum_Med_DALI_Pir/Rum_5_450/Visualization_4_330_1_1_1_1_2_1_1_1_3_1.TcVIS
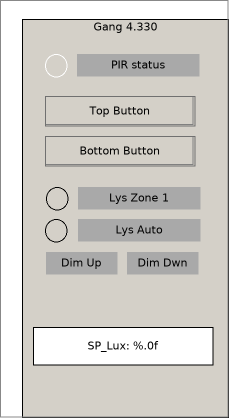
VISUALIZATION Visualization_4_330_1_1_1_1_2_1_1_1_3_1  // 229x418
    RoundedRectangle (22,19 207x399), "Gang 4.330"
    Rectangle (33,327 180x38), "SP_Lux: %.0f", text variable: P_Gang_5_135A.arrfbLysGruppe[1].fbLightCtrl.fLuxZone1
    Button (45,96 150x30), "Top Button"
        tap P_Gang_5_135A.bTopButtonZone1_Visu
    Button (45,136 150x30), "Bottom Button"
        tap P_Gang_5_135A.bBottomButtonZone1_Visu
    Ellipse (46,187 22x23), colour toggle: P_Gang_5_135A.fbLys.fbLightCtrl.bOnZone1
    Rectangle (78,187 122x22), "Lys Zone 1"
    Rectangle (46,252 71x22), "Dim Up", colour toggle: P_Gang_5_135A.arrfbLysGruppe[1].fbLightCtrl.bDimUp
    Rectangle (127,252 71x22), "Dim Dwn", colour toggle: P_Gang_5_135A.arrfbLysGruppe[1].fbLightCtrl.bDimDwn
    Ellipse (45,219 22x23), colour toggle: P_Gang_5_135A.arrfbLysGruppe[1].fbLightCtrl.bAutoZone1
    Rectangle (78,219 122x22), "Lys Auto"
    Ellipse (45,54 22x23), colour toggle: P_Gang_5_135A.arrfbLysGruppe[1].fbLightCtrl.bPIR
    Rectangle (77,54 122x22), "PIR status"
END_VISUALIZATION

// ---- POUs/Alle_Rum/Rum_Med_DALI_Pir/Rum_5_448B/Visualization_4_330_1_1_1_1_2_1.TcVIS
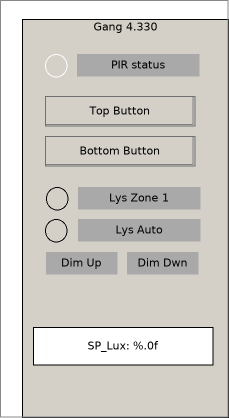
VISUALIZATION Visualization_4_330_1_1_1_1_2_1  // 229x418
    RoundedRectangle (22,19 207x399), "Gang 4.330"
    Rectangle (33,327 180x38), "SP_Lux: %.0f", text variable: P_Gang_5_135A.arrfbLysGruppe[1].fbLightCtrl.fLuxZone1
    Button (45,96 150x30), "Top Button"
        tap P_Gang_5_135A.bTopButtonZone1_Visu
    Button (45,136 150x30), "Bottom Button"
        tap P_Gang_5_135A.bBottomButtonZone1_Visu
    Ellipse (46,187 22x23), colour toggle: P_Gang_5_135A.fbLys.fbLightCtrl.bOnZone1
    Rectangle (78,187 122x22), "Lys Zone 1"
    Rectangle (46,252 71x22), "Dim Up", colour toggle: P_Gang_5_135A.arrfbLysGruppe[1].fbLightCtrl.bDimUp
    Rectangle (127,252 71x22), "Dim Dwn", colour toggle: P_Gang_5_135A.arrfbLysGruppe[1].fbLightCtrl.bDimDwn
    Ellipse (45,219 22x23), colour toggle: P_Gang_5_135A.arrfbLysGruppe[1].fbLightCtrl.bAutoZone1
    Rectangle (78,219 122x22), "Lys Auto"
    Ellipse (45,54 22x23), colour toggle: P_Gang_5_135A.arrfbLysGruppe[1].fbLightCtrl.bPIR
    Rectangle (77,54 122x22), "PIR status"
END_VISUALIZATION

// ---- POUs/Alle_Rum/Rum_Med_DALI_Pir/Rum_5_450B/Visualization_4_330_1_1_1_1_2_1_1_1_3_1_1_1_1.TcVIS
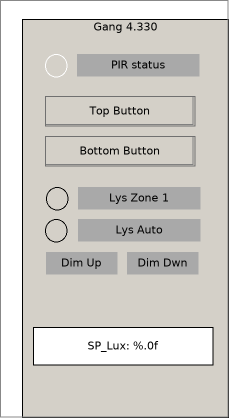
VISUALIZATION Visualization_4_330_1_1_1_1_2_1_1_1_3_1_1_1_1  // 229x418
    RoundedRectangle (22,19 207x399), "Gang 4.330"
    Rectangle (33,327 180x38), "SP_Lux: %.0f", text variable: P_Gang_5_135A.arrfbLysGruppe[1].fbLightCtrl.fLuxZone1
    Button (45,96 150x30), "Top Button"
        tap P_Gang_5_135A.bTopButtonZone1_Visu
    Button (45,136 150x30), "Bottom Button"
        tap P_Gang_5_135A.bBottomButtonZone1_Visu
    Ellipse (46,187 22x23), colour toggle: P_Gang_5_135A.fbLys.fbLightCtrl.bOnZone1
    Rectangle (78,187 122x22), "Lys Zone 1"
    Rectangle (46,252 71x22), "Dim Up", colour toggle: P_Gang_5_135A.arrfbLysGruppe[1].fbLightCtrl.bDimUp
    Rectangle (127,252 71x22), "Dim Dwn", colour toggle: P_Gang_5_135A.arrfbLysGruppe[1].fbLightCtrl.bDimDwn
    Ellipse (45,219 22x23), colour toggle: P_Gang_5_135A.arrfbLysGruppe[1].fbLightCtrl.bAutoZone1
    Rectangle (78,219 122x22), "Lys Auto"
    Ellipse (45,54 22x23), colour toggle: P_Gang_5_135A.arrfbLysGruppe[1].fbLightCtrl.bPIR
    Rectangle (77,54 122x22), "PIR status"
END_VISUALIZATION

// ---- POUs/Alle_Rum/Rum_Med_DALI_Pir/Rum_5_441A/Visualization_5_338_1_1_2_1_1_1_1_1_1_1_1_1_1_1_1_2_2_2.TcVIS
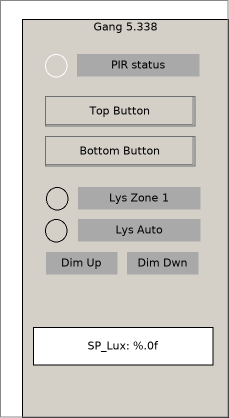
VISUALIZATION Visualization_5_338_1_1_2_1_1_1_1_1_1_1_1_1_1_1_1_2_2_2  // 229x418
    RoundedRectangle (22,19 207x399), "Gang 5.338"
    Rectangle (33,327 180x38), "SP_Lux: %.0f", text variable: P_Gang_5_338.arrfbLysGruppe[1].fbLightCtrl.fLuxZone1
    Button (45,96 150x30), "Top Button"
        tap P_Gang_5_338.bTopButtonZone1_Visu
    Button (45,136 150x30), "Bottom Button"
        tap P_Gang_5_338.bBottomButtonZone1_Visu
    Ellipse (46,187 22x23), colour toggle: P_Gang_5_338.arrfbLysGruppe[1].fbLightCtrl.bOnZone1
    Rectangle (78,187 122x22), "Lys Zone 1"
    Rectangle (46,252 71x22), "Dim Up", colour toggle: P_Gang_5_338.arrfbLysGruppe[1].fbLightCtrl.bDimUp
    Rectangle (127,252 71x22), "Dim Dwn", colour toggle: P_Gang_5_338.arrfbLysGruppe[1].fbLightCtrl.bDimDwn
    Ellipse (45,219 22x23), colour toggle: P_Gang_5_338.arrfbLysGruppe[1].fbLightCtrl.bAutoZone1
    Rectangle (78,219 122x22), "Lys Auto"
    Ellipse (45,54 22x23), colour toggle: P_Gang_5_338.arrfbLysGruppe[1].fbLightCtrl.bPIR
    Rectangle (77,54 122x22), "PIR status"
END_VISUALIZATION

// ---- POUs/DALI/DALI_Setup/VISUs/Visu_DALICommissioning.TcVIS
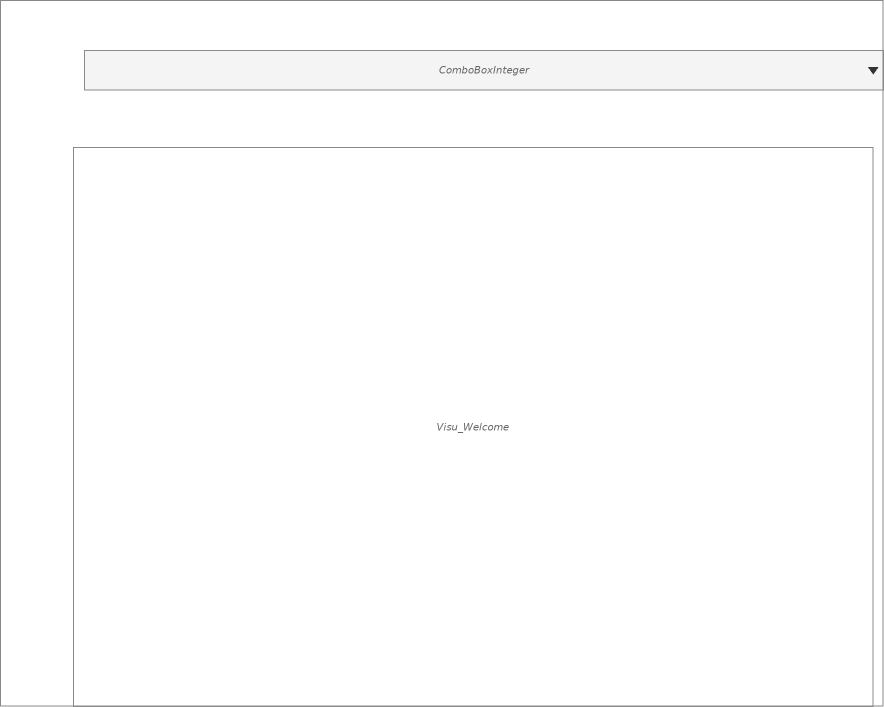
VISUALIZATION Visu_DALICommissioning  // 884x707
    ComboBoxInteger (84,50 800x40), variable: DALI_Commissioning.nSelectedDialog, input disabled if: DALI_Commissioning.bDisableComboBox, text list: 'TextList_Dialogs'
    Frame (73,147 800x560), frame switch variable: DALI_Commissioning.nSelectedDialog
        shows Visu_Welcome()
        shows Visu_Part102Commands()
        shows Visu_Part102Addressing()
        shows Visu_Part102Parameters()
        shows Visu_Part102Groups()
        shows Visu_Part102Scenes()
        shows Visu_Part102MemoryBank()
        shows Visu_Part102SetFading()
        shows Visu_Part202()
        shows Visu_Part205()
        shows Visu_Part207()
        shows Visu_Part208Switching()
        shows Visu_Part103Addressing()
        shows Visu_Part103Parameters()
        shows Visu_Part103Identify()
        shows Visu_Part301PushButton()
        shows Visu_Part302AbsoluteInputDevice()
        shows Visu_Part303OccupancySensor()
        shows Visu_Part304LightSensor()
        shows Visu_Part300GenericDevice()
        shows Visu_Part103MemoryBank()
        shows Visu_KL6821Configuration()
END_VISUALIZATION

// ---- POUs/DALI/DALI_Setup/VISUs/Visu_DALICommissioning/Visu_Part102Addressing.TcVIS
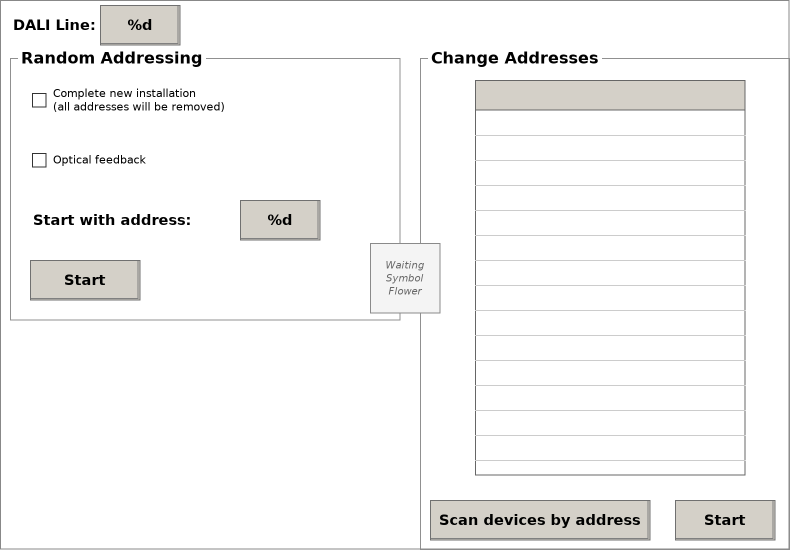
VISUALIZATION Visu_Part102Addressing  // 790x550
    GroupBox (420,50 370x500), "Change Addresses"
        Table (55,30 270x395), data array: DALI_Commissioning.fbPart102Addressing.aChangeAddressList
            p3854506369: DALI_Commissioning.fbPart102Addressing.aChangeAddressList[INDEX].nOldAddress
            p1892666644: DALI_Commissioning.fbPart102Addressing.aChangeAddressList[INDEX].nNewAddress
            p338671338: DALI_Commissioning.fbPart102Addressing.aChangeAddressList[INDEX].nRandomAddress
            p2170511999: DALI_Commissioning.fbPart102Addressing.aChangeAddressList[INDEX].nErrors
            Columns.Column.[0].Template: DALI_Commissioning.fbPart102Addressing.aNoShortAddress[INDEX]
            Columns.Column.[1].Template: DALI_Commissioning.fbPart102Addressing.aNoShortAddress[INDEX]; OnMouseClick: write the text variable via Default, min 0, max 63, title "New Short Address"
        Button (255,450 100x40), "Start"
            OnMouseClick: execute { DALI_Commissioning.fbPart102Addressing.bStartChangeAddress := TRUE; }
        Button (10,450 220x40), "Scan devices by address"
            OnMouseClick: execute { DALI_Commissioning.fbPart102Addressing.bScanDevices := TRUE; }
    GroupBox (10,50 390x270), "Random Addressing"
        Button (20,210 110x40), "Start"
            OnMouseClick: execute { DALI_Commissioning.fbPart102Addressing.bStartRandomAddressing := TRUE; }
        Checkbox (20,30 360x40), "Complete new installation (all addresses will be removed)", variable: DALI_Commissioning.fbPart102Addressing.bNewInstallation
        Checkbox (20,90 360x40), "Optical feedback", variable: DALI_Commissioning.fbPart102Addressing.bOpticalFeedback
        Textfield (20,150 200x40), "Start with address:"
        Button (230,150 80x40), "%d", text variable: DALI_Commissioning.fbPart102Addressing.nStartAddress
            OnMouseClick: write the text variable via Default, min 0, max 63, title "Insert Short Address"
    WaitingSymbolFlower (370,243 70x70), invisible if: DALI_Commissioning.fbPart102Addressing.bHideWaitSymbol
    Group (10,5 170x40)
        Textfield (0,0 110x40), "DALI Line:"
        Button (90,0 80x40), "%d", text variable: GVL_Internal.nDALILine
            OnMouseClick: write the text variable via Default, min 1, max 10, title "Choose line"
END_VISUALIZATION

// ---- POUs/DALI/DALI_Setup/VISUs/Visu_DALICommissioning/Visu_Part103Addressing.TcVIS
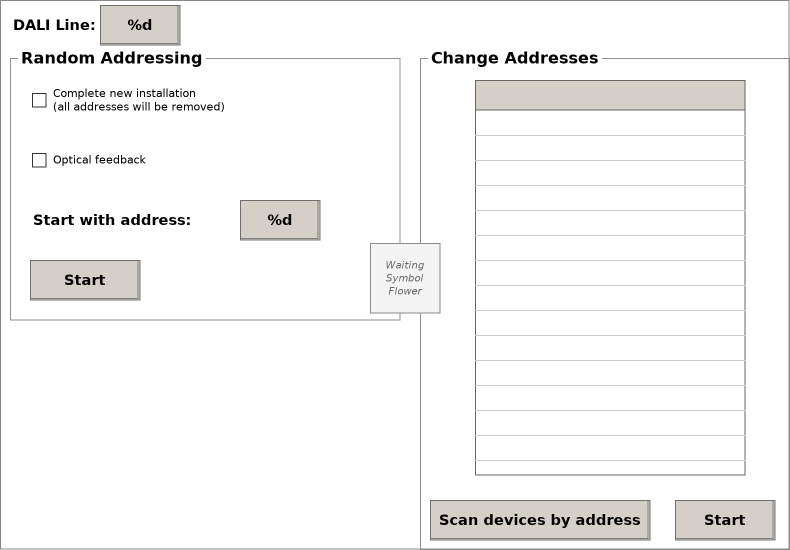
VISUALIZATION Visu_Part103Addressing  // 790x550
    GroupBox (420,50 370x500), "Change Addresses"
        Table (55,30 270x395), data array: DALI_Commissioning.fbPart103Addressing.aChangeAddressList
            p3854506369: DALI_Commissioning.fbPart103Addressing.aChangeAddressList[INDEX].nOldAddress
            p1892666644: DALI_Commissioning.fbPart103Addressing.aChangeAddressList[INDEX].nNewAddress
            p338671338: DALI_Commissioning.fbPart103Addressing.aChangeAddressList[INDEX].nRandomAddress
            p2170511999: DALI_Commissioning.fbPart103Addressing.aChangeAddressList[INDEX].nErrors
            Columns.Column.[0].Template: DALI_Commissioning.fbPart103Addressing.aNoShortAddress[INDEX]
            Columns.Column.[1].Template: DALI_Commissioning.fbPart103Addressing.aNoShortAddress[INDEX]; OnMouseClick: write the text variable via Default, min 0, max 63, title "New Short Address"
        Button (255,450 100x40), "Start"
            OnMouseClick: execute { DALI_Commissioning.fbPart103Addressing.bStartChangeAddress := TRUE; }
        Button (10,450 220x40), "Scan devices by address"
            OnMouseClick: execute { DALI_Commissioning.fbPart103Addressing.bScanDevices := TRUE; }
    GroupBox (10,50 390x270), "Random Addressing"
        Button (20,210 110x40), "Start"
            OnMouseClick: execute { DALI_Commissioning.fbPart103Addressing.bStartRandomAddressing := TRUE; }
        Checkbox (20,30 360x40), "Complete new installation (all addresses will be removed)", variable: DALI_Commissioning.fbPart103Addressing.bNewInstallation
        Checkbox (20,90 360x40), "Optical feedback", variable: DALI_Commissioning.fbPart103Addressing.bOpticalFeedback
        Textfield (20,150 200x40), "Start with address:"
        Button (230,150 80x40), "%d", text variable: DALI_Commissioning.fbPart103Addressing.nStartAddress
            OnMouseClick: write DALI_Commissioning.fbPart103Addressing.nStartAddress via Default, min 0, max 63, title "Insert Short Address"
    WaitingSymbolFlower (370,243 70x70), invisible if: DALI_Commissioning.fbPart103Addressing.bHideWaitSymbol
    Group (10,5 170x40)
        Textfield (0,0 110x40), "DALI Line:"
        Button (90,0 80x40), "%d", text variable: GVL_Internal.nDALILine
            OnMouseClick: write the text variable via Default, min 1, max 10, title "Choose line"
END_VISUALIZATION

// ---- POUs/DALI/DALI_Setup/VISUs/Visu_DALICommissioning/Visu_Part202.TcVIS
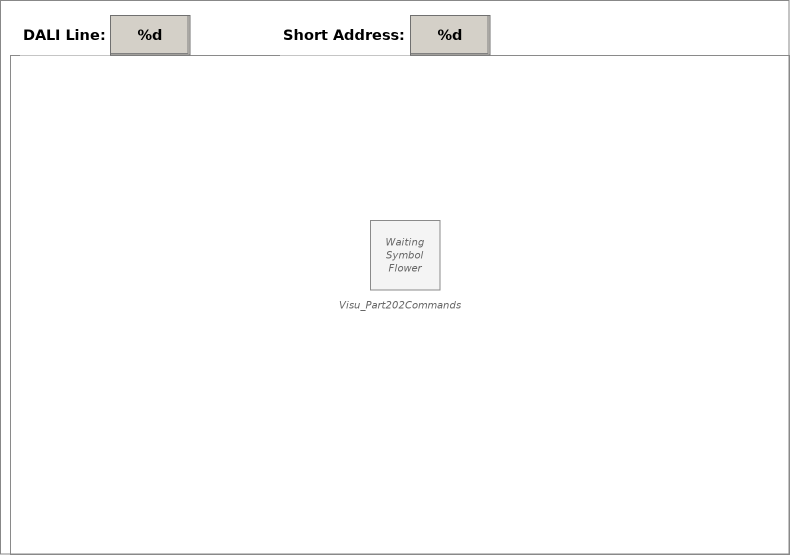
VISUALIZATION Visu_Part202  // 790x555
    TabControl (10,55 780x500)
        shows Visu_Part202Commands()
        shows Visu_Part202Status()
        shows Visu_Part202Parameters()
        [0]: TabTitle=Commands
        [1]: TabTitle=Status
        [2]: TabTitle=Parameters
    Group (280,15 210x40)
        Textfield (0,0 130x40), "Short Address:"
        Button (130,0 80x40), "%d", text variable: DALI_Commissioning.fbPart202Emergency.nAddress
            OnMouseClick: write the text variable via Default, min 0, max 63, title "Insert Short Address"
    Group (20,15 170x40)
        Textfield (0,0 110x40), "DALI Line:"
        Button (90,0 80x40), "%d", text variable: GVL_Internal.nDALILine
            OnMouseClick: write the text variable via Default, min 1, max 10, title "Choose line"
    WaitingSymbolFlower (370,220 70x70), invisible if: DALI_Commissioning.fbPart202Emergency.bHideWaitSymbol
END_VISUALIZATION

// ---- POUs/DALI/DALI_Setup/VISUs/Visu_DALICommissioning/Visu_Part303OccupancySensor.TcVIS
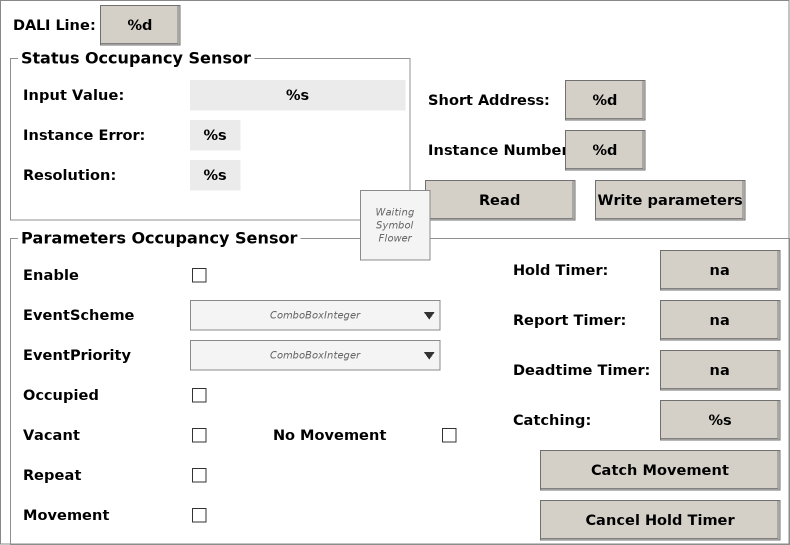
VISUALIZATION Visu_Part303OccupancySensor  // 790x545
    GroupBox (10,230 780x315), "Parameters Occupancy Sensor"
        Button (650,70 120x40), "%d s", text variable: DALI_Commissioning.fbPart303OccupancySensor.nReport
            OnMouseClick: write the text variable via Default, min 0, max 255, title "Insert value for report timer"
        Button (650,70 120x40), "na", invisible if: Not DALI_Commissioning.fbPart303OccupancySensor.bNoReportTimer, input disabled if: Not DALI_Commissioning.fbPart303OccupancySensor.bNoReportTimer
        Textfield (500,125 145x30), "Deadtime Timer:"
        Textfield (500,75 145x30), "Report Timer:"
        Textfield (500,25 145x30), "Hold Timer:"
        Button (650,20 120x40), "%d s", text variable: DALI_Commissioning.fbPart303OccupancySensor.nHold, invisible if: DALI_Commissioning.fbPart303OccupancySensor.bNoHoldTimer, input disabled if: DALI_Commissioning.fbPart303OccupancySensor.bNoHoldTimer
            OnMouseClick: write the text variable via Default, min 0, max 2538, title "Insert value for hold timer"
        Textfield (10,30 150x30), "Enable"
        Button (650,120 120x40), "%d ms", text variable: DALI_Commissioning.fbPart303OccupancySensor.nDeadtime
            OnMouseClick: write the text variable via Default, min 0, max 12750, title "Insert value for deadtime timer"
        Checkbox (180,30 30x30), variable: DALI_Commissioning.fbPart303OccupancySensor.bEnable
        Textfield (10,70 150x30), "EventScheme"
        Textfield (10,150 150x30), "Occupied"
        Textfield (10,190 150x30), "Vacant"
        Textfield (10,230 150x30), "Repeat"
        Textfield (10,270 150x30), "Movement"
        Textfield (260,190 150x30), "No Movement"
        Checkbox (180,150 30x30), variable: DALI_Commissioning.fbPart303OccupancySensor.bOccupied
        Checkbox (180,190 30x30), variable: DALI_Commissioning.fbPart303OccupancySensor.bVacant
        Checkbox (180,230 30x30), variable: DALI_Commissioning.fbPart303OccupancySensor.bRepeat
        Checkbox (430,190 30x30), variable: DALI_Commissioning.fbPart303OccupancySensor.bNoMovement
        ComboBoxInteger (180,70 250x30), variable: DALI_Commissioning.fbPart303OccupancySensor.eEventScheme, text list: 'EventScheme'
        Checkbox (180,270 30x30), variable: DALI_Commissioning.fbPart303OccupancySensor.bMovement
        Button (650,120 120x40), "na", invisible if: Not DALI_Commissioning.fbPart303OccupancySensor.bNoDeadtimeTimer, input disabled if: Not DALI_Commissioning.fbPart303OccupancySensor.bNoDeadtimeTimer
        Button (530,270 240x40), "Cancel Hold Timer"
            OnMouseClick: execute { DALI_Commissioning.fbPart303OccupancySensor.bCancelHoldTimer := true; }
        Textfield (10,110 150x30), "EventPriority"
        ComboBoxInteger (180,110 250x30), variable: DALI_Commissioning.fbPart303OccupancySensor.eEventPriority, text list: 'EventPriority'
        Button (650,20 120x40), "na", invisible if: Not DALI_Commissioning.fbPart303OccupancySensor.bNoHoldTimer, input disabled if: Not DALI_Commissioning.fbPart303OccupancySensor.bNoHoldTimer
        Button (530,220 240x40), "Catch Movement"
            OnMouseClick: execute { DALI_Commissioning.fbPart303OccupancySensor.bCatchMovement := true; }
        Textfield (500,175 145x30), "Catching:"
    GroupBox (10,50 400x170), "Status Occupancy Sensor"
        Textfield (10,30 160x30), "Input Value:"
        Textfield (10,70 160x30), "Instance Error:"
        Textfield (10,110 160x30), "Resolution:"
        Textfield (180,30 215x30), "%s", text variable: DALI_Commissioning.fbPart303OccupancySensor.sInputValue
        Textfield (180,70 50x30), "%s", text variable: DALI_Commissioning.fbPart303OccupancySensor.nInstanceError
        Textfield (180,110 50x30), "%s", text variable: DALI_Commissioning.fbPart303OccupancySensor.nResolution
    Button (425,180 150x40), "Read"
        OnMouseClick: execute { DALI_Commissioning.fbPart303OccupancySensor.bRead := TRUE; }
    WaitingSymbolFlower (360,190 70x70), invisible if: DALI_Commissioning.fbPart303OccupancySensor.bHideWaitSymbol
    Button (595,180 150x40), "Write parameters"
        OnMouseClick: execute { DALI_Commissioning.fbPart303OccupancySensor.bWrite := TRUE; }
    Button (660,400 120x40), "%s", text variable: DALI_Commissioning.fbPart303OccupancySensor.sCatching
        OnMouseClick: write the text variable via Default, min 0, max 12750, title "Insert value for deadtime timer"
    Group (10,5 170x40)
        Textfield (0,0 110x40), "DALI Line:"
        Button (90,0 80x40), "%d", text variable: GVL_Internal.nDALILine
            OnMouseClick: write the text variable via Default, min 1, max 10, title "Choose line"
    Textfield (425,80 130x40), "Short Address:"
    Button (565,80 80x40), "%d", text variable: DALI_Commissioning.fbPart303OccupancySensor.nAddress
        OnMouseClick: write the text variable via Default, min 0, max 63, title "Insert Short Address"
    Textfield (425,130 150x40), "Instance Number:"
    Button (565,130 80x40), "%d", text variable: DALI_Commissioning.fbPart303OccupancySensor.nInstanceAddress
        OnMouseClick: write the text variable via Default, min 0, max 31, title "Insert instance number"
END_VISUALIZATION
